Staubli VAL3: stop.pgx

public program stop()
begin
  resetMotion()
end
